FUNCTION_BLOCK FB_Testmaschinentuer
VAR_INPUT
	bVentil	: BOOL;
END_VAR
VAR_OUTPUT
	bDoorC	: BOOL;
	bDoorO	: BOOL;
END_VAR
VAR
	fbTon_O	: TON;
	fbTon_C	: TON;
	tDuration : TIME := T#5S;
END_VAR

fbTon_C(IN:= bVentil, PT:= tDuration, Q=> , ET=> );
fbTon_O(IN:= NOT bVentil, PT:= tDuration, Q=> , ET=> );

IF bVentil THEN
	bDoorO := FALSE;
	
	IF fbTon_C.Q THEN
		bDoorC := TRUE;
	END_IF
ELSIF NOT bVentil THEN
	bDoorC := FALSE;

	IF fbTon_O.Q THEN
		bDoorO := TRUE;
	END_IF
END_IF

END_FUNCTION_BLOCK

(* stored: Version 1.1.0.1, ProductVersion 3.1.4024.15
   POU FB_Testmaschinentuer: Id {3cd13bc1-8cc2-48e0-b308-67082b0854ce}, SpecialFunc None *)
